(* CoDeSys 2.3.9.37 project: Cap11_6.pro *)
(* Libraries: Standard.lib 4.10.05 12:14:46, IecSfc.lib 13.4.06 16:51:28 *)

(* POU PLC_PRG, SFC *)
PROGRAM PLC_PRG
VAR
       (* Entradas *)
	A: BOOL;
	B: BOOL;
       (* Salidas*)
	Salida: BOOL;
       (* Otras *)
       FinSubred:BOOL;
END_VAR
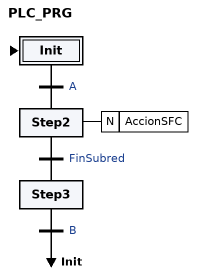
INITIAL_STEP Init:
END_STEP
TRANSITION FROM Init TO Step2 := A;
END_TRANSITION
STEP Step2:
	AccionSFC(N);
END_STEP
TRANSITION FROM Step2 TO Step3 := FinSubred;
END_TRANSITION
STEP Step3:
END_STEP
TRANSITION FROM Step3 TO Init := B;
END_TRANSITION
END_PROGRAM
ACTION AccionSFC:
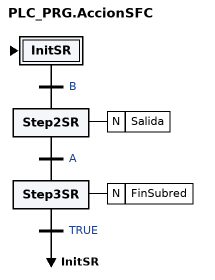
INITIAL_STEP InitSR:
END_STEP
TRANSITION FROM InitSR TO Step2SR := B;
END_TRANSITION
STEP Step2SR:
	Salida(N);
END_STEP
TRANSITION FROM Step2SR TO Step3SR := A;
END_TRANSITION
STEP Step3SR:
	FinSubred(N);
END_STEP
TRANSITION FROM Step3SR TO InitSR := TRUE;
END_TRANSITION
END_ACTION

(* Visualisation Visu
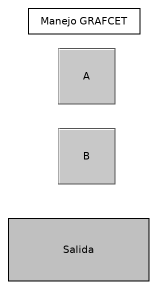
button at (80,50)-(137,106): text "A"; taps PLC_PRG.A
button at (80,130)-(137,186): text "B"; taps PLC_PRG.B
rectangle at (50,10)-(162,36): text "Manejo GRAFCET"
rounded rectangle at (30,220)-(171,283): text "Salida"; alarm colour if PLC_PRG.Salida
*)
